(* CODESYS project WashingMachineSim.export

Project tree, tasks and I/O mapping:
  program Simulation_Program [ST]
*)

// Simulation_Program
PROGRAM Simulation_Program
VAR
		bulls_eye_open_past	:BOOL := TRUE;
END_VAR

(*Temperature value simulation*)
IF ((GVL.hot)AND(NOT GVL.heat_fail)) THEN 
	GVL.temperature := GVL.temperature + 1;
ELSE
	GVL.temperature := GVL.temperature - 1;
END_IF

IF GVL.temperature > 100 THEN 
	GVL.temperature := 100;
END_IF

IF GVL.temperature < 0 THEN 
	GVL.temperature := 0;
END_IF


(*Soap level simulation*)
IF GVL.fillsoap THEN 
	GVL.soaplevel := GVL.soaplevel + 5;
ELSIF GVL.emptysoap THEN 
	GVL.soaplevel := GVL.soaplevel - 3;
END_IF

IF GVL.soaplevel >= 50 THEN 
	GVL.soaplevel := 50;
	GVL.fillsoap := FALSE;
END_IF

IF GVL.soaplevel < 0 THEN 
	GVL.soaplevel := 0;
END_IF


(*Door state simulation*)
IF ((GVL.bulls_eye_open <> bulls_eye_open_past)AND(NOT GVL.bulls_eye_lock)) THEN 
	bulls_eye_open_past := GVL.bulls_eye_open ;
ELSIF GVL.bulls_eye_lock THEN
	GVL.bulls_eye_open := bulls_eye_open_past;
END_IF


(*Water level simulation*)
IF ((GVL.fillwater)AND(NOT GVL.water_in_fail)) THEN 
	GVL.waterlevel := GVL.waterlevel + 2;
ELSIF ((GVL.emptywater)AND(NOT GVL.water_out_fail)) THEN
	GVL.waterlevel := GVL.waterlevel - 4;
END_IF

IF GVL.waterlevel > 150 THEN 
	GVL.waterlevel := 150;
END_IF

IF GVL.waterlevel < 0 THEN 
	GVL.waterlevel := 0;
END_IF


(*Motor simulation*)
IF (GVL.motor_on) THEN 
	GVL.motor := GVL.motor + 10;
END_IF

IF GVL.motor > 360 THEN 
	GVL.motor := 0;
END_IF

END_PROGRAM
